FUNCTION_BLOCK FB_LinearActuator
VAR
    // STATE & CONFIGURATION
    eState      : ENUM_LinearActuatorState := LAS_LinearActuator_Uninitialised;
    tTimeout    : TIME := T#10S;

    // ERROR HANDLING
    bError      : BOOL;
    sErrorMsg   : STRING(80);
	bHoldDriveFaulted : BOOL;
	
    // REFERENCES
    pActuator   : POINTER TO ST_LinearActuator;

    // EDGE SELECTION FLAGS 
    bProxInRisingEdge   : BOOL := TRUE;   
    bProxOutRisingEdge  : BOOL := TRUE;  
    bProx2RisingEdge    : BOOL := TRUE;    
    bProx3RisingEdge    : BOOL := TRUE;  
    bFirstCycle : BOOL := TRUE;
	
    // EDGE DETECTION TRIGGERS
    r_trig_proxIn   : R_TRIG;             
    f_trig_proxIn   : F_TRIG;            
    r_trig_proxOut  : R_TRIG;            
    f_trig_proxOut  : F_TRIG;            
    r_trig_prox2    : R_TRIG;
    f_trig_prox2    : F_TRIG;
    r_trig_prox3    : R_TRIG;
    f_trig_prox3    : F_TRIG;
    
    // HELPER VARIABLES
    bIsGui   : BOOL;  
	bIsCmp   : BOOL;
    bIsBasic      : BOOL;  
    bDetectError : BOOL;
	
    // EDGE DETECTION RESULTS
    bProxInDetected     : BOOL;
    bProxOutDetected    : BOOL;
    bProx2Detected      : BOOL;
    bProx3Detected      : BOOL;

END_VAR

METHOD CheckDriveFault : BOOL
VAR
	pAlarmCondition : POINTER TO BOOL;
END_VAR
IF NOT bIsBasic THEN
	pAlarmCondition := F_GetLinearActuatorAlarmCondition(pActuator^.sName, 'DriveFaulted');
	
    IF pActuator^.bFaultDI^ := TRUE THEN
		IF NOT bHoldDriveFaulted THEN
			eState := LAS_LinearActuator_Error;
		END_IF
		
		bHoldDriveFaulted := TRUE;
		IF pAlarmCondition <> 0 THEN
			pAlarmCondition^ := TRUE;
		END_IF
	ELSE
		IF pAlarmCondition <> 0 THEN
			pAlarmCondition^ := FALSE;
		END_IF
	END_IF
END_IF
END_METHOD

METHOD Extend : INT
VAR
    pAlarmCondition : POINTER TO BOOL;
	nStop : INT;
END_VAR
Extend := 0;

//CheckDriveFault();
UpdateProxDetection();

IF bFirstCycle THEN
	GetPosition();
	bFirstCycle := FALSE;
END_IF

CASE eState OF
    LAS_LinearActuator_Retracted, LAS_LinearActuator_Error: //Allow Linear Actuator movement when position is unknown
        SetForwardMovement();
		pActuator^.tTimeout(IN := TRUE, PT := tTimeout);
        eState := LAS_LinearActuator_Extending;
        
    LAS_LinearActuator_AtProx2, LAS_LinearActuator_AtProx3:
        pActuator^.bFwdDO^ := TRUE;
        pActuator^.bBckwDO^ := FALSE;
        eState := LAS_LinearActuator_Extending;

    LAS_LinearActuator_Extending:
		pActuator^.tTimeout(IN := TRUE, PT := tTimeout);
		
		IF bCriticalAlarm THEN
			pActuator^.tTimeout(IN := FALSE);
            Stop(); 
			//bHoldDriveFaulted := FALSE;
			bFirstCycle := TRUE;
            Extend := -1;
		END_IF
		
		IF bIsBasic THEN
			SetForwardMovement(); //Continuous call of basic linear actuators
		END_IF
		
		IF bProx2Detected THEN
			IF bIsGui THEN
				eState := LAS_LinearActuator_AtProx2;
			ELSIF bIsCmp THEN
				eState := LAS_LinearActuator_Error;		
				pAlarmCondition := F_GetLinearActuatorAlarmCondition(pActuator^.sName, 'UnknownPosition');
				IF pAlarmCondition <> 0 THEN
					pAlarmCondition^ := TRUE;
				END_IF
				
				Stop();
				pActuator^.tTimeout(IN := FALSE);
				bHoldDriveFaulted := FALSE;
				bFirstCycle := TRUE;
				Extend := -1; 
			END_IF
		ELSIF bProx3Detected THEN
			eState := LAS_LinearActuator_AtProx3;

			IF pActuator^.bSpeedControlDO <> 0 THEN
				pActuator^.bSpeedControlDO^ := TRUE;  // Slow down when reaching Prox3
			END_IF
		END_IF
		
        IF bProxOutDetected THEN
			Stop();
			
			eState := LAS_LinearActuator_Extended;
			bHoldDriveFaulted := FALSE;
			bFirstCycle := TRUE;
            Extend := 1; 
		    pActuator^.tTimeout(IN := FALSE);
        END_IF
        
        IF pActuator^.tTimeout.Q THEN // Check for timeout
            eState := LAS_LinearActuator_Error;
            
            pAlarmCondition := F_GetLinearActuatorAlarmCondition(pActuator^.sName, 'MotionTimedOut');
            IF pAlarmCondition <> 0 THEN
                pAlarmCondition^ := TRUE;
            END_IF
            
			pActuator^.tTimeout(IN := FALSE);
            Stop(); 
			bHoldDriveFaulted := FALSE;
			bFirstCycle := TRUE;
            Extend := -1;
        END_IF

    LAS_LinearActuator_Extended:
        Extend := 1; // Already extended
		
		bFirstCycle := TRUE;
		pActuator^.tTimeout(IN := FALSE);
END_CASE
END_METHOD

METHOD FB_Init: BOOL
VAR_INPUT
    bInitRetains: BOOL;
    bInCopyCode: BOOL;   
    Actuator : POINTER TO ST_LinearActuator;  
END_VAR
VAR
    pAlarmCondition : POINTER TO BOOL;
END_VAR
pActuator := Actuator;
bHoldDriveFaulted := FALSE;

(* Detect actuator type *)
bIsGui := pActuator^.sName = 'HeatExCoupola3' OR pActuator^.sName = 'RegenCoupola3';
bIsCmp := pActuator^.sName = 'Compressor1' OR pActuator^.sName = 'Compressor3';
bIsBasic := NOT bIsGui AND NOT bIsCmp;

(* Initialise speed control to fast *)
IF bIsGui THEN
    pActuator^.bSpeedControlDO^ := FALSE; 
END_IF

(* Initialise stop to false *)
IF NOT bIsBasic THEN
	pActuator^.bStopControlDO^ := FALSE; 
END_IF

//GetPosition();
END_METHOD

METHOD GetPosition : BOOL
VAR
	pAlarmCondition : POINTER TO BOOL;
END_VAR
VAR_OUTPUT
	State : SINT;
END_VAR
bDetectError := FALSE;
UpdateProxDetection();

IF bProxInRisingEdge = pActuator^.bProxIn^ THEN    
    eState := LAS_LinearActuator_Retracted;
    State := 0;  
	GetPosition := TRUE;
	bDetectError := TRUE;

ELSIF bProxOutRisingEdge = pActuator^.bProxOut^ THEN
    eState := LAS_LinearActuator_Extended;
    State := 1;  
	GetPosition := TRUE;
	bDetectError := TRUE;
END_IF

IF bIsGui AND NOT bDetectError THEN
	IF bProx2RisingEdge = pActuator^.bProx2^ THEN
		eState := LAS_LinearActuator_AtProx2;
		State := 2;  
		GetPosition := TRUE;
		bDetectError := TRUE;
	ELSIF bProx3RisingEdge = pActuator^.bProx3^ THEN
		eState := LAS_LinearActuator_AtProx3;
		State := 3;  
		GetPosition := TRUE;
		bDetectError := TRUE;
	END_IF
END_IF

IF NOT bDetectError THEN
	eState := LAS_LinearActuator_Error;
	
	pAlarmCondition := F_GetLinearActuatorAlarmCondition(pActuator^.sName, 'UnknownPosition');
	IF pAlarmCondition <> 0 THEN
		pAlarmCondition^ := TRUE;
	END_IF

	State := -1;
	GetPosition := FALSE;
END_IF
END_METHOD

METHOD Home : INT
VAR
    pAlarmCondition : POINTER TO BOOL;
	nStop : INT;
END_VAR
Home := 0;

//CheckDriveFault();
UpdateProxDetection();

IF bFirstCycle THEN
	GetPosition();
	bFirstCycle := FALSE;
END_IF

CASE eState OF
    LAS_LinearActuator_Extended, LAS_LinearActuator_Error: //Allow Linear Actuator movement when position is unknown
        SetBackwardMovement();
		pActuator^.tTimeout(IN := TRUE, PT := tTimeout);
        eState := LAS_LinearActuator_Retracting;

    LAS_LinearActuator_AtProx3, LAS_LinearActuator_AtProx2:
        pActuator^.bFwdDO^ := FALSE;
        pActuator^.bBckwDO^ := TRUE;
        eState := LAS_LinearActuator_Retracting;

    LAS_LinearActuator_Retracting:
		IF bCriticalAlarm THEN
			pActuator^.tTimeout(IN := FALSE);
            Stop(); 
			//bHoldDriveFaulted := FALSE;
			bFirstCycle := TRUE;
            Home := -1;
		END_IF
		
		pActuator^.tTimeout(IN := TRUE, PT := tTimeout);
		
		IF bIsBasic THEN
			SetBackwardMovement(); //Continuous call of basic linear actuators
		END_IF
		
        IF bIsGui THEN
            IF bProx3Detected THEN
                eState := LAS_LinearActuator_AtProx3;
            ELSIF bProx2Detected THEN
                eState := LAS_LinearActuator_AtProx2;

                IF pActuator^.bSpeedControlDO <> 0 THEN
                    pActuator^.bSpeedControlDO^ := TRUE;  // Slow down when reaching Prox2
                END_IF
            END_IF
        END_IF
        
        IF bProxInDetected THEN
			Stop();
			
			eState := LAS_LinearActuator_Retracted;
			bHoldDriveFaulted := FALSE;
			bFirstCycle := TRUE;
            Home := 1; 
		    pActuator^.tTimeout(IN := FALSE);
        END_IF
        
        // Check for timeout
        IF pActuator^.tTimeout.Q THEN
            eState := LAS_LinearActuator_Error;
            pActuator^.tTimeout(IN := FALSE);
			
            pAlarmCondition := F_GetLinearActuatorAlarmCondition(pActuator^.sName, 'MotionTimedOut');
            IF pAlarmCondition <> 0 THEN
                pAlarmCondition^ := TRUE;
            END_IF
            
            pActuator^.tTimeout(IN := FALSE);
            Stop(); 
			bHoldDriveFaulted := FALSE;
			bFirstCycle := TRUE;
            Home := -1;
        END_IF

    LAS_LinearActuator_Retracted:
        Home := 1; 
		bFirstCycle := TRUE;
		pActuator^.tTimeout(IN := FALSE);
END_CASE
END_METHOD

METHOD Reset : BOOL
VAR
    i : UINT;
    sActuatorName : STRING(50);
	pAlarmCondition : POINTER TO BOOL;
END_VAR
VAR_OUTPUT
    State : SINT;
END_VAR
sActuatorName := pActuator^.sName;

//CheckDriveFault();

IF GetPosition(State => State) THEN
	pAlarmCondition := F_GetLinearActuatorAlarmCondition(pActuator^.sName, 'UnknownPosition');
	IF pAlarmCondition <> 0 THEN
		pAlarmCondition^ := FALSE;
	END_IF
	
	pAlarmCondition := F_GetLinearActuatorAlarmCondition(pActuator^.sName, 'MotionTimedOut');
	IF pAlarmCondition <> 0 THEN
		pAlarmCondition^ := FALSE;
	END_IF
END_IF
END_METHOD

METHOD SetBackwardMovement : BOOL
VAR_INPUT
END_VAR
pActuator^.bFwdDO^ := FALSE;
pActuator^.bBckwDO^ := TRUE;
END_METHOD

METHOD SetForwardMovement : BOOL
pActuator^.bFwdDO^ := TRUE;
pActuator^.bBckwDO^ := FALSE;
END_METHOD

METHOD Stop : INT

VAR_OUTPUT
	State : SINT;
END_VAR
//CheckDriveFault();

pActuator^.bFwdDO^ := FALSE;
pActuator^.bBckwDO^ := FALSE;
pActuator^.tTimeout(IN := FALSE);

IF NOT bIsBasic THEN
	pActuator^.bStopControlDO^ := TRUE;
END_IF

GetPosition(State => State);
END_METHOD

METHOD UpdateProxDetection : BOOL
r_trig_proxIn(CLK := pActuator^.bProxIn^);
f_trig_proxIn(CLK := pActuator^.bProxIn^);
r_trig_proxOut(CLK := pActuator^.bProxOut^);
f_trig_proxOut(CLK := pActuator^.bProxOut^);

(* Select which edge is valid based on configuration flags *)
bProxInDetected := (bProxInRisingEdge AND r_trig_proxIn.Q) OR (NOT bProxInRisingEdge AND f_trig_proxIn.Q);
bProxOutDetected := (bProxOutRisingEdge AND r_trig_proxOut.Q) OR (NOT bProxOutRisingEdge AND f_trig_proxOut.Q);

IF NOT bIsBasic THEN
    r_trig_prox2(CLK := pActuator^.bProx2^);
    f_trig_prox2(CLK := pActuator^.bProx2^);
	
	bProx2Detected := (bProx2RisingEdge AND r_trig_prox2.Q) OR (NOT bProx2RisingEdge AND f_trig_prox2.Q);
	
	IF bIsGui THEN
		r_trig_prox3(CLK := pActuator^.bProx3^);
    	f_trig_prox3(CLK := pActuator^.bProx3^);
      
    	bProx3Detected := (bProx3RisingEdge AND r_trig_prox3.Q) OR (NOT bProx3RisingEdge AND f_trig_prox3.Q);
	END_IF
END_IF
END_METHOD

END_FUNCTION_BLOCK

(* stored: Version 1.1.0.1, ProductVersion 3.1.4026.11
   POU FB_LinearActuator: Id {7b9c3bff-54cb-4df9-8ad3-e1094e9996e8}, SpecialFunc None
   Method CheckDriveFault: Id {fa98b561-2deb-4912-871f-79363f500ba9}
   Method Extend: Id {afb44406-33a7-4c96-9c8b-3094883b11ba}
   Method FB_Init: Id {70258f52-1024-4f1a-abb0-a262de844735}
   Method GetPosition: Id {0399b1b7-cdd3-4ec3-9edf-6a45105de5e5}
   Method Home: Id {f928c3cc-e926-4d68-aa06-e49d712546af}
   Method Reset: Id {ecdda1b9-dec3-446e-af49-02346c123f36}
   Method SetBackwardMovement: Id {2c497243-ee6e-4e97-99a2-fe8b03e246e5}
   Method SetForwardMovement: Id {75e1c4ab-755e-4c46-b900-5237b95878fd}
   Method Stop: Id {fb95bc7a-c6f6-46a4-ad31-adc69398fdb2}
   Method UpdateProxDetection: Id {6e178de4-6a01-4e7a-9cb7-df152934fa89} *)
